// TIA Portal V17 export
// export: Created 2023-12-22T15:28:29.8084386Z, ExportSetting WithDefaults, DisplayName Totally Integrated Automation Portal, DisplayVersion V17, DisplayName TIA Portal Openness, DisplayVersion V17, DisplayName TIA Portal Version Control Interface, DisplayVersion V17, DisplayName STEP 7 Professional, DisplayVersion V17, DisplayName STEP 7 Safety, DisplayVersion V17, DisplayName WinCC Advanced, DisplayVersion V17
FUNCTION "FC_DRV_Start" : Void   // FC100, LAD
{ S7_Optimized_Access := 'FALSE' }
VERSION : 0.1
// stored: AutoNumber false, IsIECCheckEnabled false, SetENOAutomatically false, UDAEnableTagReadback false
BEGIN

REGION Network 1: Системное время
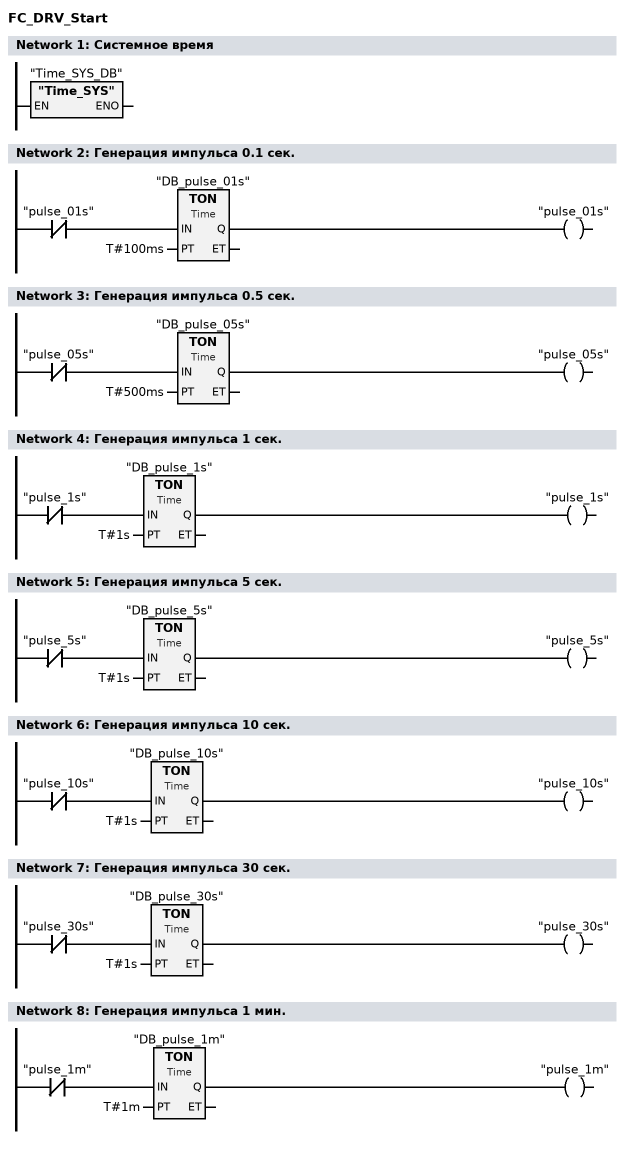
   RUNG wire#powerrail
      "Time_SYS_DB"()
   END_RUNG
   // the same network as SCL:
   "Time_SYS_DB"();   // "Time_SYS"
END_REGION

REGION Network 2: Генерация импульса 0.1 сек.
   RUNG wire#powerrail
      I_Contact( "pulse_01s" )
      { S7_Templates := "time_type := Time" } "DB_pulse_01s".TON(pt := T#100ms, et =>)
      Coil( "pulse_01s" )
   END_RUNG
   // the same network as SCL:
   "DB_pulse_01s".TON(IN := NOT "pulse_01s", PT := T#100ms);
   "pulse_01s" := "DB_pulse_01s".Q;
END_REGION

REGION Network 3: Генерация импульса 0.5 сек.
   RUNG wire#powerrail
      I_Contact( "pulse_05s" )
      { S7_Templates := "time_type := Time" } "DB_pulse_05s".TON(pt := T#500ms, et =>)
      Coil( "pulse_05s" )
   END_RUNG
   // the same network as SCL:
   "DB_pulse_05s".TON(IN := NOT "pulse_05s", PT := T#500ms);
   "pulse_05s" := "DB_pulse_05s".Q;
END_REGION

REGION Network 4: Генерация импульса 1 сек.
   RUNG wire#powerrail
      I_Contact( "pulse_1s" )
      { S7_Templates := "time_type := Time" } "DB_pulse_1s".TON(pt := T#1s, et =>)
      Coil( "pulse_1s" )
   END_RUNG
   // the same network as SCL:
   "DB_pulse_1s".TON(IN := NOT "pulse_1s", PT := T#1s);
   "pulse_1s" := "DB_pulse_1s".Q;
END_REGION

REGION Network 5: Генерация импульса 5 сек.
   RUNG wire#powerrail
      I_Contact( "pulse_5s" )
      { S7_Templates := "time_type := Time" } "DB_pulse_5s".TON(pt := T#1s, et =>)
      Coil( "pulse_5s" )
   END_RUNG
   // the same network as SCL:
   "DB_pulse_5s".TON(IN := NOT "pulse_5s", PT := T#1s);
   "pulse_5s" := "DB_pulse_5s".Q;
END_REGION

REGION Network 6: Генерация импульса 10 сек.
   RUNG wire#powerrail
      I_Contact( "pulse_10s" )
      { S7_Templates := "time_type := Time" } "DB_pulse_10s".TON(pt := T#1s, et =>)
      Coil( "pulse_10s" )
   END_RUNG
   // the same network as SCL:
   "DB_pulse_10s".TON(IN := NOT "pulse_10s", PT := T#1s);
   "pulse_10s" := "DB_pulse_10s".Q;
END_REGION

REGION Network 7: Генерация импульса 30 сек.
   RUNG wire#powerrail
      I_Contact( "pulse_30s" )
      { S7_Templates := "time_type := Time" } "DB_pulse_30s".TON(pt := T#1s, et =>)
      Coil( "pulse_30s" )
   END_RUNG
   // the same network as SCL:
   "DB_pulse_30s".TON(IN := NOT "pulse_30s", PT := T#1s);
   "pulse_30s" := "DB_pulse_30s".Q;
END_REGION

REGION Network 8: Генерация импульса 1 мин.
   RUNG wire#powerrail
      I_Contact( "pulse_1m" )
      { S7_Templates := "time_type := Time" } "DB_pulse_1m".TON(pt := T#1m, et =>)
      Coil( "pulse_1m" )
   END_RUNG
   // the same network as SCL:
   "DB_pulse_1m".TON(IN := NOT "pulse_1m", PT := T#1m);
   "pulse_1m" := "DB_pulse_1m".Q;
END_REGION
END_FUNCTION
